{attribute addProperty BoxType "EL3423-0000-0016"}
{attribute addProperty Id "Unbalance_Guard_WarningAT %I*BOOL811Unbalance_Guard_ErrorAT %I*BOOL812"}
{attribute addProperty CRC "4238643945"}
{attribute addProperty SizeInBites "16"}
{attribute addProperty SizeInBytes "2"}
TYPE Total_Advanced_FCA492E9 :
STRUCT
	{attribute addProperty Name "Unbalance_Guard_Warning"}
	Unbalance_Guard_Warning AT %I* : BOOL;
	{attribute addProperty Name "Unbalance_Guard_Error"}
	Unbalance_Guard_Error AT %I* : BOOL;
END_STRUCT
END_TYPE

(* stored: Version 1.2.0.0, ProductVersion 3.1.4024.9
   DUT Total_Advanced_FCA492E9: Id {d5298ced-9b20-4a35-9d3e-cca0661dd1d8} *)
